Fanuc KAREL source: compact_preamble.KL

PROGRAM KB00127
%NOLOCKGROUP
VAR
P1 : STRING[80];P2:INTEGER;RESULT:INTEGER
BEGIN
P1='A'
P2=1
RESULT=ORD(P1,P2)
END KB00127
